Fanuc KAREL source: IO0061.KL

PROGRAM IO0061
%NOLOCKGROUP
ROUTINE RTEST
VAR
  I : INTEGER
  STATUS : INTEGER
  ENTRY : INTEGER
  A : ARRAY[3] OF INTEGER
  B : BOOLEAN
  R : REAL
  P : XYZWPR
  JPOS : JOINTPOS
  PF : POSITION
BEGIN
  I = 1
  A[1] = 2
  B = TRUE
  R = 1.0
  GOUT[I + 1] = 1
END RTEST
BEGIN
  RTEST
END IO0061
